// Mitsubishi GX Works2 project: CTrinhMayChat-Z   PLC: FX1N/FX1NC

PROGRAM MAIN
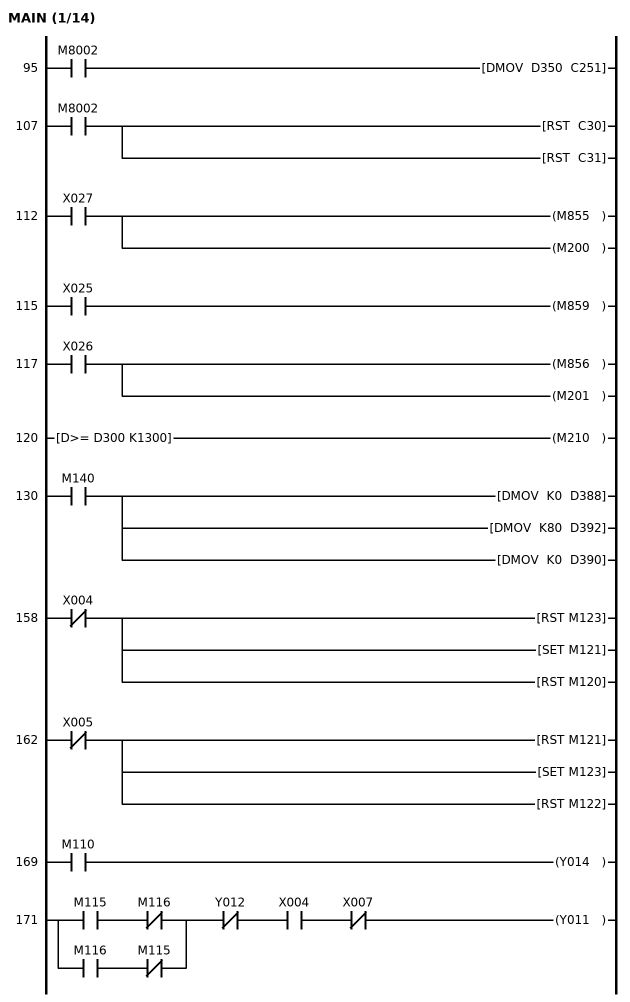
95    LD      M8002
      DMOV    D350 C251
107   LD      M8002
      RST     C30
      RST     C31
112   LD      X027
      OUT     M855
      OUT     M200
115   LD      X025
      OUT     M859
117   LD      X026
      OUT     M856
      OUT     M201
120   LDD>=   D300 K1300
      OUT     M210
130   LD      M140
      DMOV    K0 D388
      DMOV    K80 D392
      DMOV    K0 D390
158   LDI     X004
      RST     M123
      SET     M121
      RST     M120
162   LDI     X005
      RST     M121
      SET     M123
      RST     M122
169   LD      M110
      OUT     Y014
171   LD      M115
      ANI     M116
      LD      M116
      ANI     M115
      ORB
      ANI     Y012
      AND     X004
      ANI     X007
      OUT     Y011
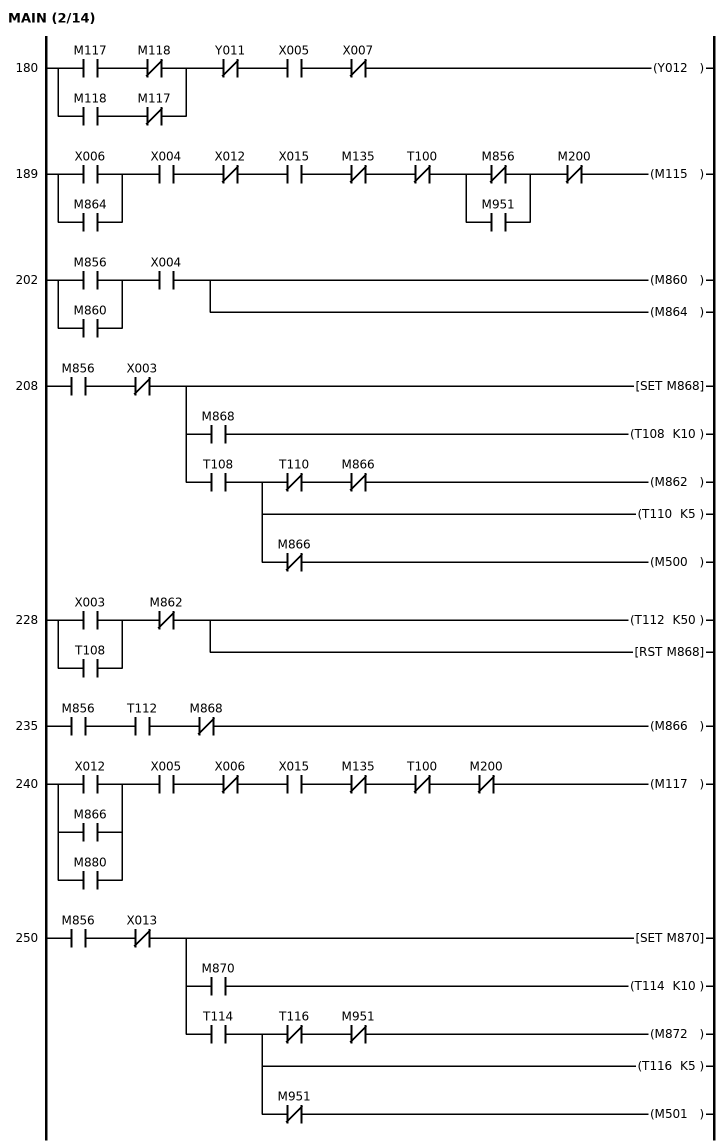
180   LD      M117
      ANI     M118
      LD      M118
      ANI     M117
      ORB
      ANI     Y011
      AND     X005
      ANI     X007
      OUT     Y012
189   LD      X006
      OR      M864
      AND     X004
      ANI     X012
      AND     X015
      ANI     M135
      ANI     T100
      LDI     M856
      OR      M951
      ANB
      ANI     M200
      OUT     M115
202   LD      M856
      OR      M860
      AND     X004
      OUT     M860
      OUT     M864
208   LD      M856
      ANI     X003
      SET     M868
      MPS
      AND     M868
      OUT     T108 K10
      MPP
      AND     T108
      MPS
      ANI     T110
      ANI     M866
      OUT     M862
      MPP
      OUT     T110 K5
      ANI     M866
      OUT     M500
228   LD      X003
      OR      T108
      ANI     M862
      OUT     T112 K50
      RST     M868
235   LD      M856
      AND     T112
      ANI     M868
      OUT     M866
240   LD      X012
      OR      M866
      OR      M880
      AND     X005
      ANI     X006
      AND     X015
      ANI     M135
      ANI     T100
      ANI     M200
      OUT     M117
250   LD      M856
      ANI     X013
      SET     M870
      MPS
      AND     M870
      OUT     T114 K10
      MPP
      AND     T114
      MPS
      ANI     T116
      ANI     M951
      OUT     M872
      MPP
      OUT     T116 K5
      ANI     M951
      OUT     M501
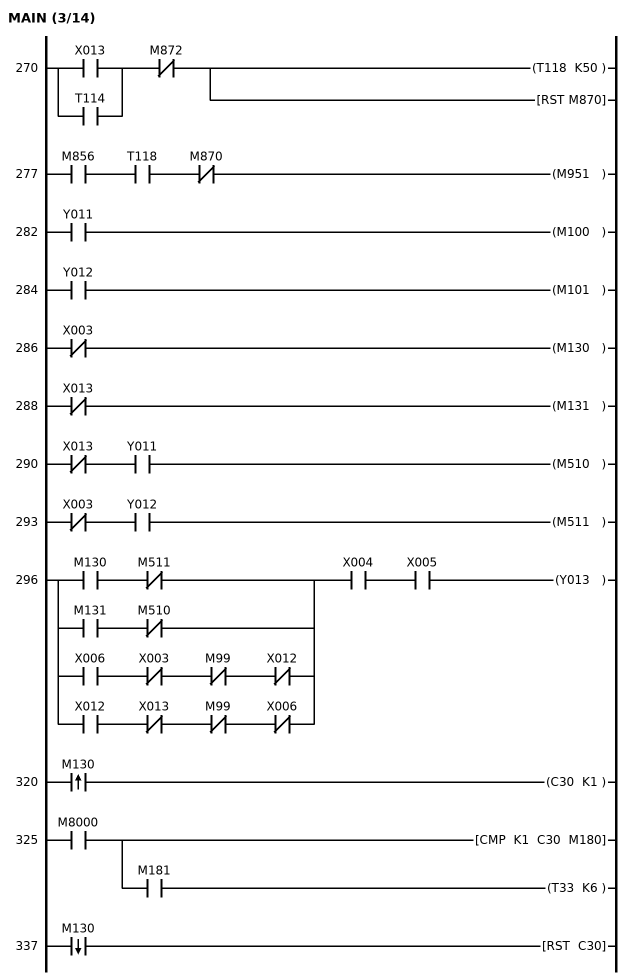
270   LD      X013
      OR      T114
      ANI     M872
      OUT     T118 K50
      RST     M870
277   LD      M856
      AND     T118
      ANI     M870
      OUT     M951
282   LD      Y011
      OUT     M100
284   LD      Y012
      OUT     M101
286   LDI     X003
      OUT     M130
288   LDI     X013
      OUT     M131
290   LDI     X013
      AND     Y011
      OUT     M510
293   LDI     X003
      AND     Y012
      OUT     M511
296   LD      M130
      ANI     M511
      LD      M131
      ANI     M510
      ORB
      LD      X006
      ANI     X003
      ANI     M99
      ANI     X012
      ORB
      LD      X012
      ANI     X013
      ANI     M99
      ANI     X006
      ORB
      AND     X004
      AND     X005
      OUT     Y013
320   LDP     M130
      OUT     C30 K1
325   LD      M8000
      CMP     K1 C30 M180
      AND     M181
      OUT     T33 K6
337   LDF     M130
      RST     C30
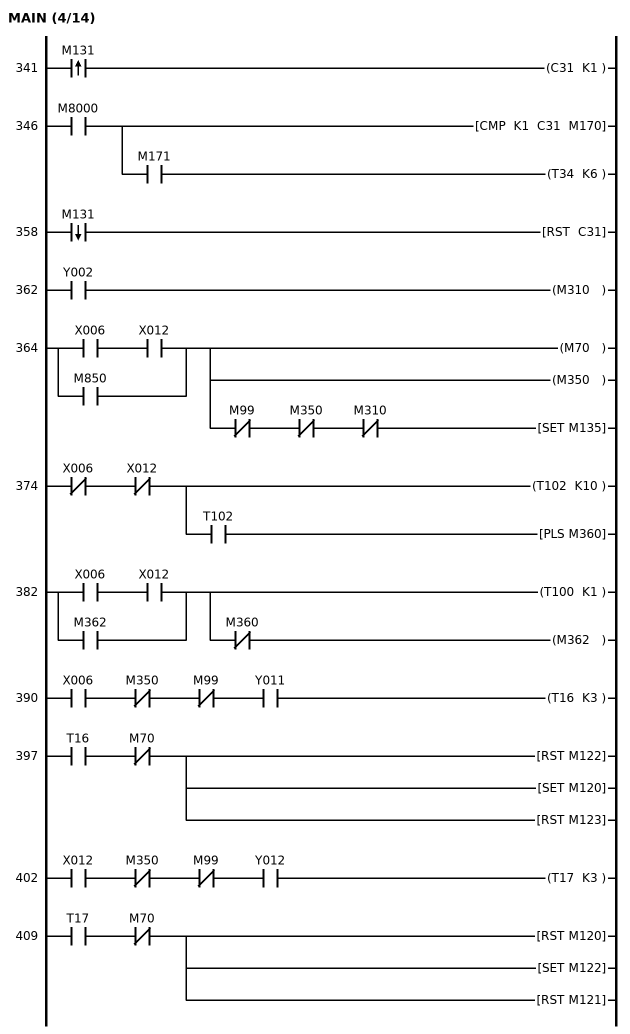
341   LDP     M131
      OUT     C31 K1
346   LD      M8000
      CMP     K1 C31 M170
      AND     M171
      OUT     T34 K6
358   LDF     M131
      RST     C31
362   LD      Y002
      OUT     M310
364   LD      X006
      AND     X012
      OR      M850
      OUT     M70
      OUT     M350
      ANI     M99
      ANI     M350
      ANI     M310
      SET     M135
374   LDI     X006
      ANI     X012
      OUT     T102 K10
      AND     T102
      PLS     M360
382   LD      X006
      AND     X012
      OR      M362
      OUT     T100 K1
      ANI     M360
      OUT     M362
390   LD      X006
      ANI     M350
      ANI     M99
      AND     Y011
      OUT     T16 K3
397   LD      T16
      ANI     M70
      RST     M122
      SET     M120
      RST     M123
402   LD      X012
      ANI     M350
      ANI     M99
      AND     Y012
      OUT     T17 K3
409   LD      T17
      ANI     M70
      RST     M120
      SET     M122
      RST     M121
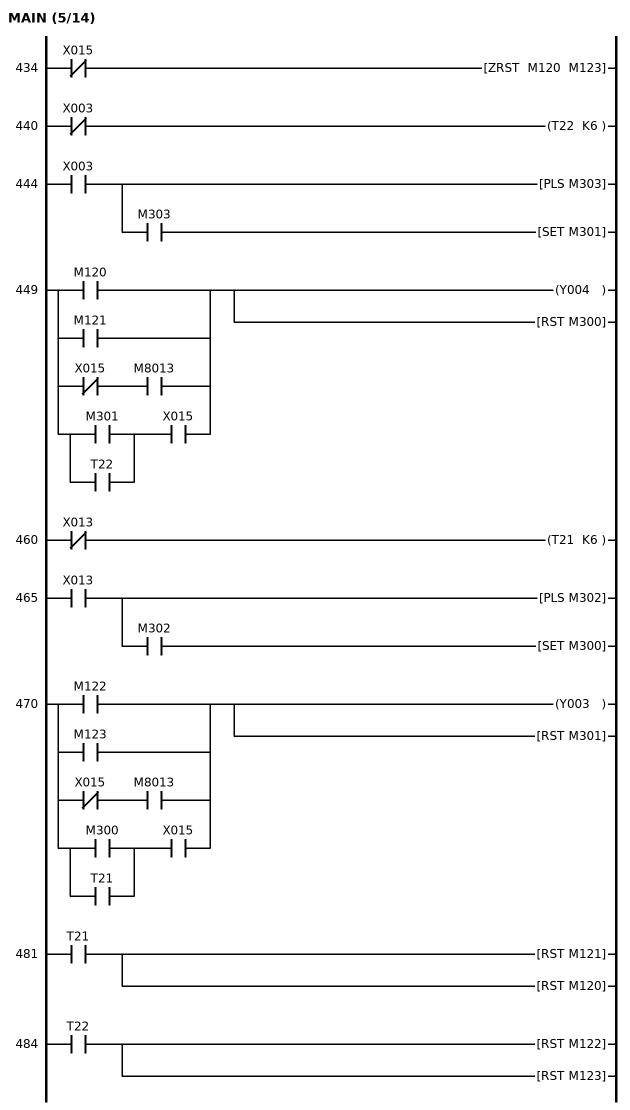
434   LDI     X015
      ZRST    M120 M123
440   LDI     X003
      OUT     T22 K6
444   LD      X003
      PLS     M303
      AND     M303
      SET     M301
449   LD      M120
      OR      M121
      LDI     X015
      AND     M8013
      ORB
      LD      M301
      OR      T22
      AND     X015
      ORB
      OUT     Y004
      RST     M300
460   LDI     X013
      OUT     T21 K6
465   LD      X013
      PLS     M302
      AND     M302
      SET     M300
470   LD      M122
      OR      M123
      LDI     X015
      AND     M8013
      ORB
      LD      M300
      OR      T21
      AND     X015
      ORB
      OUT     Y003
      RST     M301
481   LD      T21
      RST     M121
      RST     M120
484   LD      T22
      RST     M122
      RST     M123
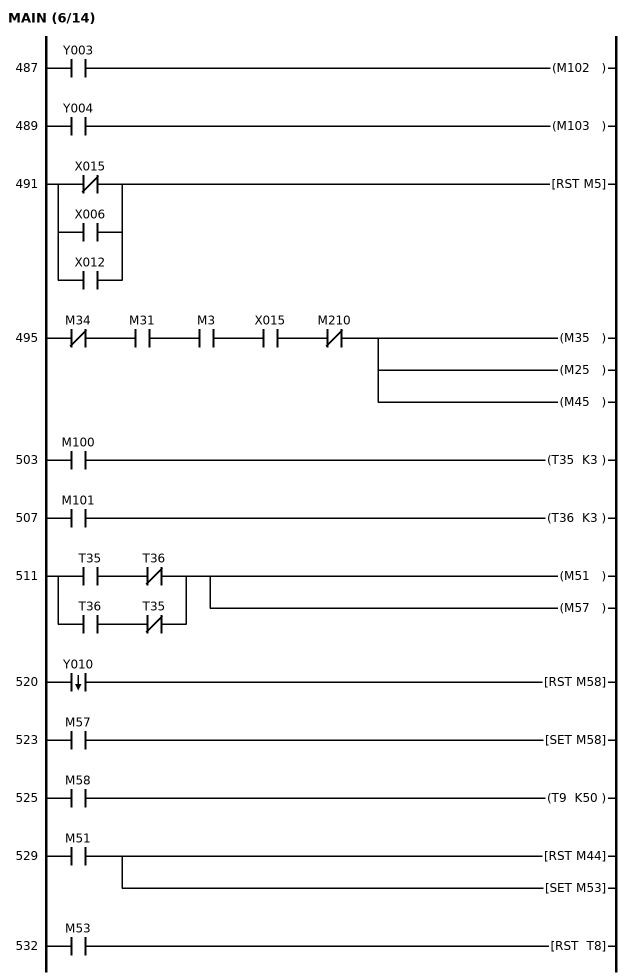
487   LD      Y003
      OUT     M102
489   LD      Y004
      OUT     M103
491   LDI     X015
      OR      X006
      OR      X012
      RST     M5
495   LDI     M34
      AND     M31
      AND     M3
      AND     X015
      ANI     M210
      OUT     M35
      OUT     M25
      OUT     M45
503   LD      M100
      OUT     T35 K3
507   LD      M101
      OUT     T36 K3
511   LD      T35
      ANI     T36
      LD      T36
      ANI     T35
      ORB
      OUT     M51
      OUT     M57
520   LDF     Y010
      RST     M58
523   LD      M57
      SET     M58
525   LD      M58
      OUT     T9 K50
529   LD      M51
      RST     M44
      SET     M53
532   LD      M53
      RST     T8
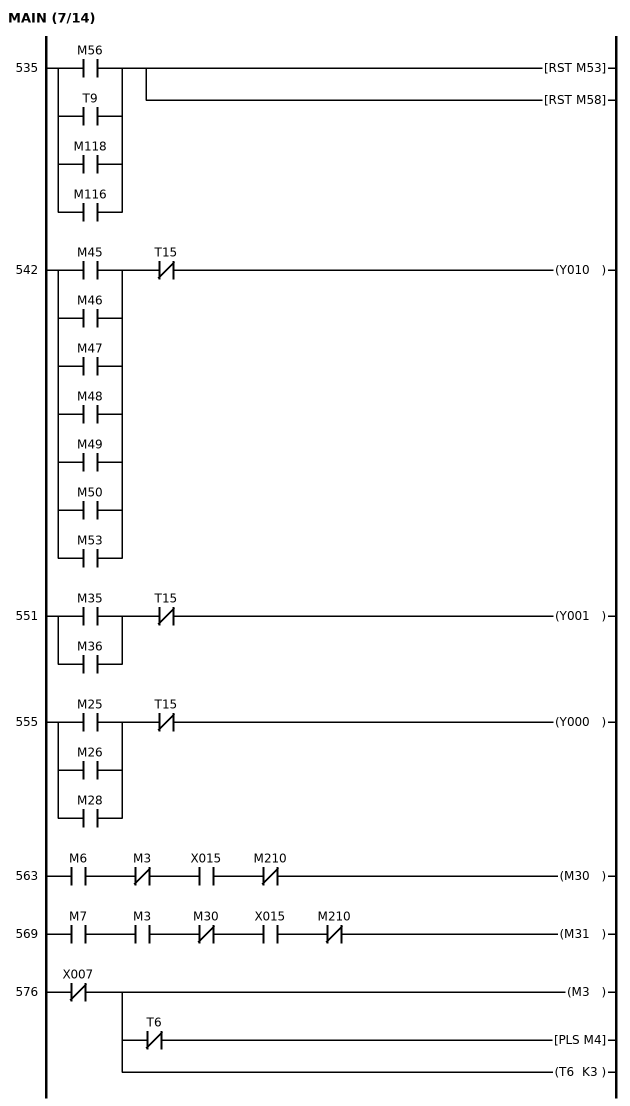
535   LD      M56
      OR      T9
      OR      M118
      OR      M116
      RST     M53
      RST     M58
542   LD      M45
      OR      M46
      OR      M47
      OR      M48
      OR      M49
      OR      M50
      OR      M53
      ANI     T15
      OUT     Y010
551   LD      M35
      OR      M36
      ANI     T15
      OUT     Y001
555   LD      M25
      OR      M26
      OR      M28
      ANI     T15
      OUT     Y000
563   LD      M6
      ANI     M3
      AND     X015
      ANI     M210
      OUT     M30
569   LD      M7
      AND     M3
      ANI     M30
      AND     X015
      ANI     M210
      OUT     M31
576   LDI     X007
      OUT     M3
      MPS
      ANI     T6
      PLS     M4
      MPP
      OUT     T6 K3
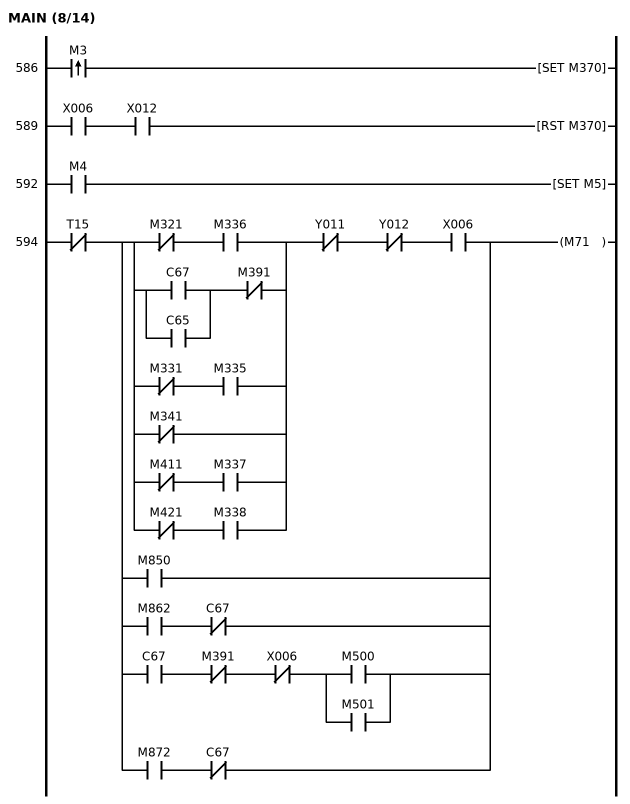
586   LDP     M3
      SET     M370
589   LD      X006
      AND     X012
      RST     M370
592   LD      M4
      SET     M5
594   LDI     T15
      LDI     M321
      AND     M336
      LD      C67
      OR      C65
      ANI     M391
      ORB
      LDI     M331
      AND     M335
      ORB
      ORI     M341
      LDI     M411
      AND     M337
      ORB
      LDI     M421
      AND     M338
      ORB
      ANI     Y011
      ANI     Y012
      AND     X006
      OR      M850
      LD      M862
      ANI     C67
      ORB
      LD      C67
      ANI     M391
      ANI     X006
      LD      M500
      OR      M501
      ANB
      ORB
      LD      M872
      ANI     C67
      ORB
      ANB
      OUT     M71
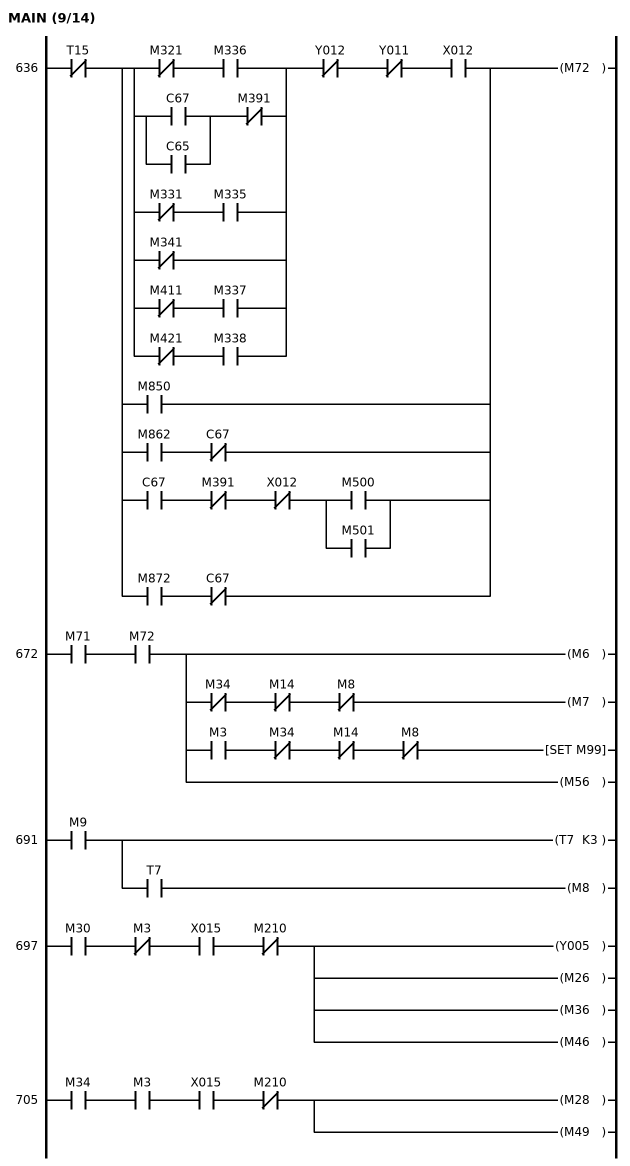
636   LDI     T15
      LDI     M321
      AND     M336
      LD      C67
      OR      C65
      ANI     M391
      ORB
      LDI     M331
      AND     M335
      ORB
      ORI     M341
      LDI     M411
      AND     M337
      ORB
      LDI     M421
      AND     M338
      ORB
      ANI     Y012
      ANI     Y011
      AND     X012
      OR      M850
      LD      M862
      ANI     C67
      ORB
      LD      C67
      ANI     M391
      ANI     X012
      LD      M500
      OR      M501
      ANB
      ORB
      LD      M872
      ANI     C67
      ORB
      ANB
      OUT     M72
672   LD      M71
      AND     M72
      OUT     M6
      MPS
      ANI     M34
      ANI     M14
      ANI     M8
      OUT     M7
      MRD
      AND     M3
      ANI     M34
      ANI     M14
      ANI     M8
      SET     M99
      MPP
      OUT     M56
691   LD      M9
      OUT     T7 K3
      AND     T7
      OUT     M8
697   LD      M30
      ANI     M3
      AND     X015
      ANI     M210
      OUT     Y005
      OUT     M26
      OUT     M36
      OUT     M46
705   LD      M34
      AND     M3
      AND     X015
      ANI     M210
      OUT     M28
      OUT     M49
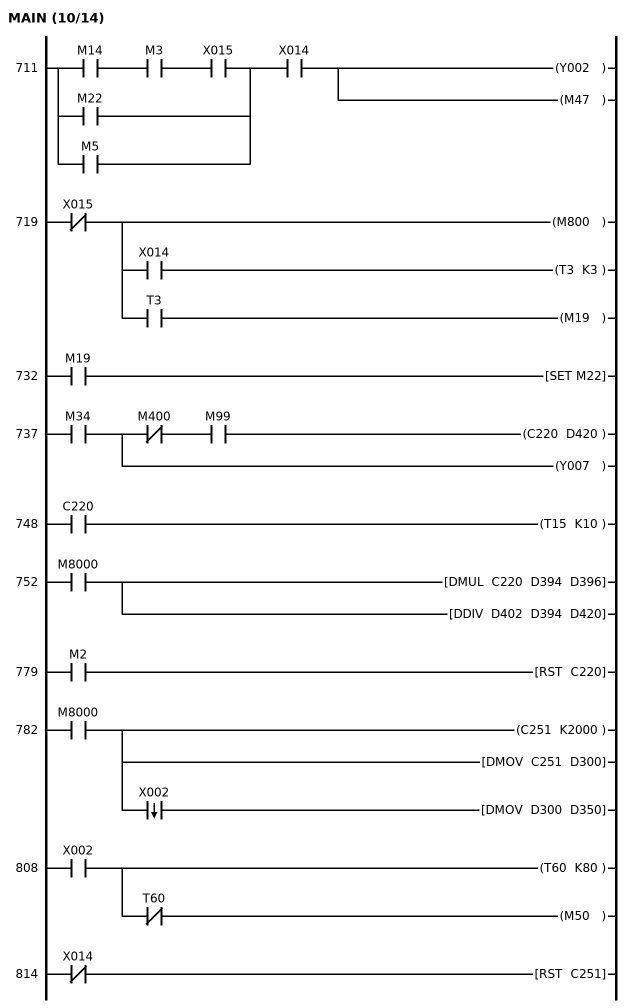
711   LD      M14
      AND     M3
      AND     X015
      OR      M22
      OR      M5
      AND     X014
      OUT     Y002
      OUT     M47
719   LDI     X015
      OUT     M800
      MPS
      AND     X014
      OUT     T3 K3
      MPP
      AND     T3
      OUT     M19
732   LD      M19
      SET     M22
737   LD      M34
      MPS
      ANI     M400
      AND     M99
      OUT     C220 D420
      MPP
      OUT     Y007
748   LD      C220
      OUT     T15 K10
752   LD      M8000
      DMUL    C220 D394 D396
      DDIV    D402 D394 D420
779   LD      M2
      RST     C220
782   LD      M8000
      OUT     C251 K2000
      DMOV    C251 D300
      ANDF    X002
      DMOV    D300 D350
808   LD      X002
      OUT     T60 K80
      ANI     T60
      OUT     M50
814   LDI     X014
      RST     C251
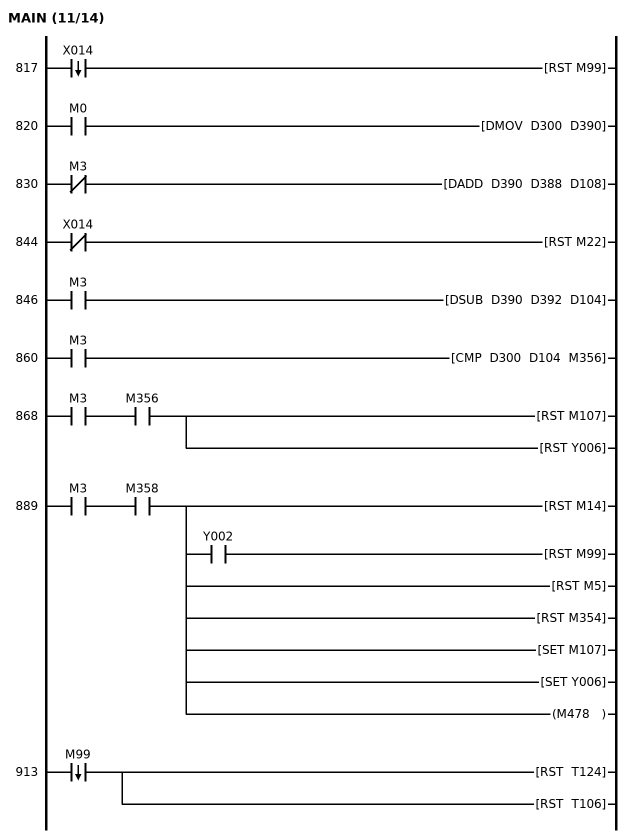
817   LDF     X014
      RST     M99
820   LD      M0
      DMOV    D300 D390
830   LDI     M3
      DADD    D390 D388 D108
844   LDI     X014
      RST     M22
846   LD      M3
      DSUB    D390 D392 D104
860   LD      M3
      CMP     D300 D104 M356
868   LD      M3
      AND     M356
      RST     M107
      RST     Y006
889   LD      M3
      AND     M358
      RST     M14
      MPS
      AND     Y002
      RST     M99
      MPP
      RST     M5
      RST     M354
      SET     M107
      SET     Y006
      OUT     M478
913   LDF     M99
      RST     T124
      RST     T106
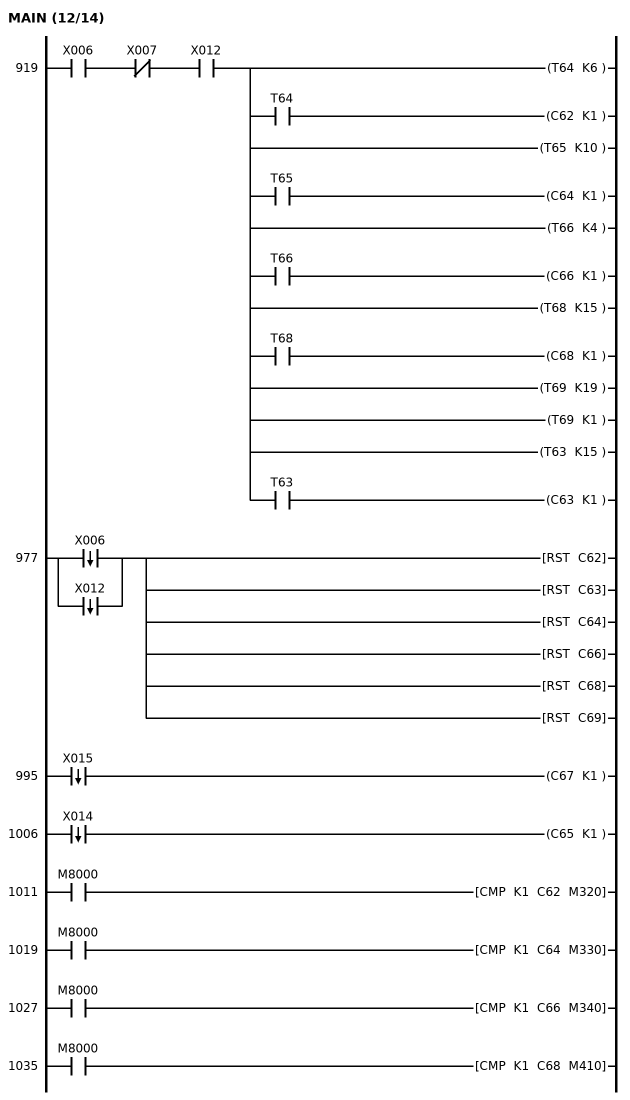
919   LD      X006
      ANI     X007
      AND     X012
      OUT     T64 K6
      MPS
      AND     T64
      OUT     C62 K1
      MPP
      OUT     T65 K10
      MPS
      AND     T65
      OUT     C64 K1
      MPP
      OUT     T66 K4
      MPS
      AND     T66
      OUT     C66 K1
      MPP
      OUT     T68 K15
      MPS
      AND     T68
      OUT     C68 K1
      MPP
      OUT     T69 K19
      OUT     T69 K1
      OUT     T63 K15
      AND     T63
      OUT     C63 K1
977   LDF     X006
      ORF     X012
      RST     C62
      RST     C63
      RST     C64
      RST     C66
      RST     C68
      RST     C69
995   LDF     X015
      OUT     C67 K1
1006  LDF     X014
      OUT     C65 K1
1011  LD      M8000
      CMP     K1 C62 M320
1019  LD      M8000
      CMP     K1 C64 M330
1027  LD      M8000
      CMP     K1 C66 M340
1035  LD      M8000
      CMP     K1 C68 M410
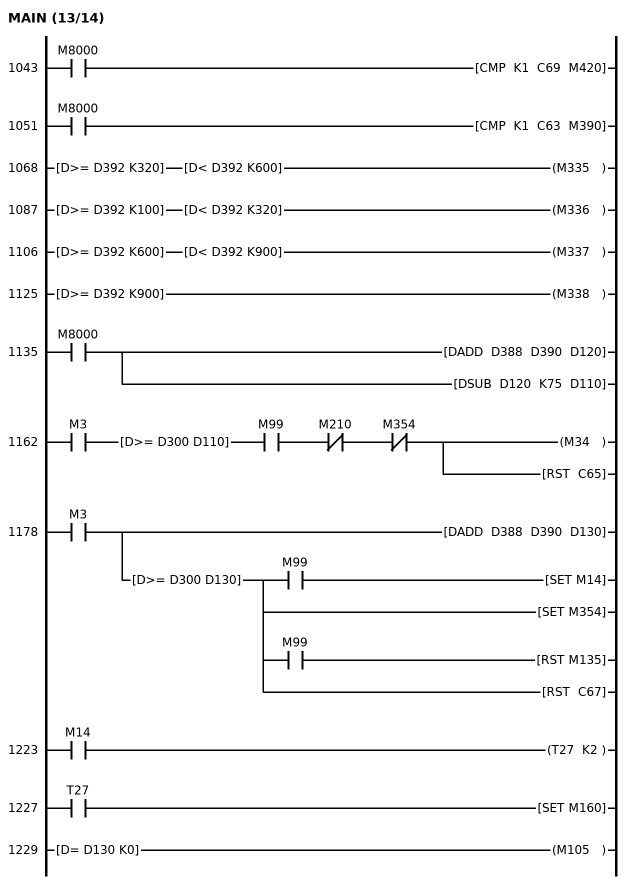
1043  LD      M8000
      CMP     K1 C69 M420
1051  LD      M8000
      CMP     K1 C63 M390
1068  LDD>=   D392 K320
      ANDD<   D392 K600
      OUT     M335
1087  LDD>=   D392 K100
      ANDD<   D392 K320
      OUT     M336
1106  LDD>=   D392 K600
      ANDD<   D392 K900
      OUT     M337
1125  LDD>=   D392 K900
      OUT     M338
1135  LD      M8000
      DADD    D388 D390 D120
      DSUB    D120 K75 D110
1162  LD      M3
      ANDD>=  D300 D110
      AND     M99
      ANI     M210
      ANI     M354
      OUT     M34
      RST     C65
1178  LD      M3
      DADD    D388 D390 D130
      ANDD>=  D300 D130
      MPS
      AND     M99
      SET     M14
      MPP
      SET     M354
      MPS
      AND     M99
      RST     M135
      MPP
      RST     C67
1223  LD      M14
      OUT     T27 K2
1227  LD      T27
      SET     M160
1229  LDD=    D130 K0
      OUT     M105
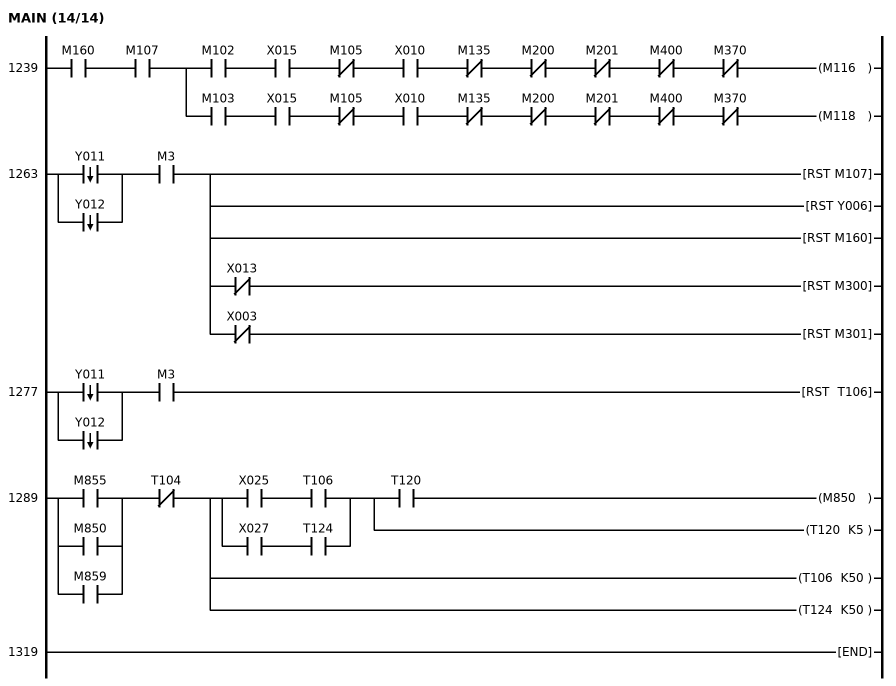
1239  LD      M160
      AND     M107
      MPS
      AND     M102
      AND     X015
      ANI     M105
      AND     X010
      ANI     M135
      ANI     M200
      ANI     M201
      ANI     M400
      ANI     M370
      OUT     M116
      MPP
      AND     M103
      AND     X015
      ANI     M105
      AND     X010
      ANI     M135
      ANI     M200
      ANI     M201
      ANI     M400
      ANI     M370
      OUT     M118
1263  LDF     Y011
      ORF     Y012
      AND     M3
      RST     M107
      RST     Y006
      RST     M160
      MPS
      ANI     X013
      RST     M300
      MPP
      ANI     X003
      RST     M301
1277  LDF     Y011
      ORF     Y012
      AND     M3
      RST     T106
1289  LD      M855
      OR      M850
      OR      M859
      ANI     T104
      MPS
      LD      X025
      AND     T106
      LD      X027
      AND     T124
      ORB
      ANB
      MPS
      AND     T120
      OUT     M850
      MPP
      OUT     T120 K5
      MPP
      OUT     T106 K50
      OUT     T124 K50
1319  END
END_PROGRAM
